Staubli VAL3: Motion.pgx

program Motion()
  local jointRx jJoint
  local bool cr
  local num idMove
begin
  //*******************************************************************************
  //*   ______
  //*  / _____) /|
  //* | |      / /
  //* | | /\  / /
  //* | | \ \/ /  _      Copyright (c) KEOLABS, 2016
  //* | |  \__/  | |        http://www.keolabs.com
  //* | |________| |
  //*  \__________/
  //*
  //********************************************************************************
  //*@file          : Motion
  //*@author        : Yves Ragot
  //*@version       : $Id: Motion.pgx 1365 2016-11-18 16:00:54Z yves $
  //*@brief         : Execute requested mouvement
  //*
  //*******************************************************************************/

  do

    wait(ExecuteMotion)

    // check if mouvement order already sent
    if (isEmpty())

        if (CartesianMode)

            // Cartesian mouvement
            cr = pointToJoint(tCurrentTool, jHome, pTargetPoint, jJoint)
            if ((isInRange(jJoint)) and (cr == true))

                restartMove()

                // launch mouvement
                if (AlignMode)
                    idMove = movel(pTargetPoint, tCurrentTool, mNomSpeed)
                else
                    idMove = movej(pTargetPoint, tCurrentTool, mNomSpeed)
                endIf

            else
                GeneralStatus = 100
                LastErrorCode = 153
            endIf

        else

          // joint mouvement
          if (isInRange(jTargetJoint))
              restartMove()
              idMove = movej(jTargetJoint, tCurrentTool, mNomSpeed)
          else
              GeneralStatus = 100
              LastErrorCode = 153
          endIf

        endIf

    // if (isEmpty())
    else
        GeneralStatus = 101
        LastErrorCode = 150
    endIf

//    if (idMove == -1)
//        GeneralStatus = 100
//        LastErrorCode = 153
//    endIf

    // if right command
    if (GeneralStatus == 0)
        // set status = busy
        GeneralStatus = 1
        MoveRunning = true
    endIf

    // wait end of mouvement if not asynchronous
    if (AsyncMode == false)
        waitEndMove()
        wait(isSettled())
    endIf

    ExecuteMotion = false

  until false

end
